// TIA Portal V20 export
FUNCTION_BLOCK "Simulation"   // FB25, LAD
// stored: MemoryReserve 100, Namespace Unit1.Em5, SetENOAutomatically false
   VAR_INPUT
      simulation { ExternalAccessible := 'False'; ExternalVisible := 'False'; ExternalWritable := 'False'} : Bool;
   END_VAR
   VAR
      instMainPnPActuator { ExternalAccessible := 'False'; ExternalVisible := 'False'; ExternalWritable := 'False'} : Array[0..9] of "LER_SimActuator";
      instAlignTableActuator { ExternalAccessible := 'False'; ExternalVisible := 'False'; ExternalWritable := 'False'} : Array[0..9] of "LER_SimActuator";
      instNgPnPActuator { ExternalAccessible := 'False'; ExternalVisible := 'False'; ExternalWritable := 'False'} : Array[0..9] of "LER_SimActuator";
   END_VAR
   VAR_TEMP   // added for the SCL form of the ladder/FBD networks
      _w1 : Bool;
   END_VAR
BEGIN

REGION Network 1: Main P&P Two Way Actuator
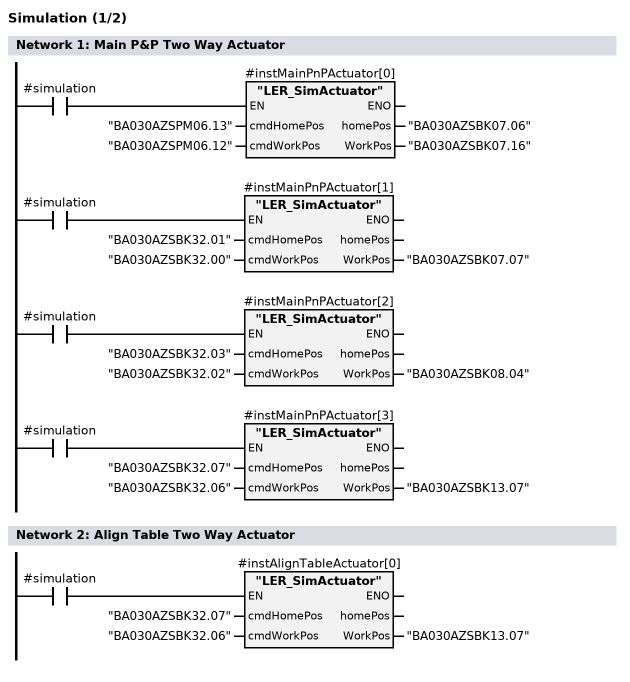
   RUNG wire#powerrail
      Contact( #simulation )
      #instMainPnPActuator[0](cmdHomePos := "BA030AZSPM06.13", cmdWorkPos := "BA030AZSPM06.12", homePos => "BA030AZSBK07.06", WorkPos => "BA030AZSBK07.16")
   END_RUNG
   RUNG wire#powerrail
      Contact( #simulation )
      #instMainPnPActuator[1](cmdHomePos := "BA030AZSBK32.01", cmdWorkPos := "BA030AZSBK32.00", homePos =>, WorkPos => "BA030AZSBK07.07")
   END_RUNG
   RUNG wire#powerrail
      Contact( #simulation )
      #instMainPnPActuator[2](cmdHomePos := "BA030AZSBK32.03", cmdWorkPos := "BA030AZSBK32.02", homePos =>, WorkPos => "BA030AZSBK08.04")
   END_RUNG
   RUNG wire#powerrail
      Contact( #simulation )
      #instMainPnPActuator[3](cmdHomePos := "BA030AZSBK32.07", cmdWorkPos := "BA030AZSBK32.06", homePos =>, WorkPos => "BA030AZSBK13.07")
   END_RUNG
   // the same network as SCL:
   IF #simulation THEN
       #instMainPnPActuator[0](cmdHomePos := "BA030AZSPM06.13",   // "LER_SimActuator"
                               cmdWorkPos := "BA030AZSPM06.12",
                               homePos => "BA030AZSBK07.06",
                               WorkPos => "BA030AZSBK07.16");
       #instMainPnPActuator[1](cmdHomePos := "BA030AZSBK32.01",   // "LER_SimActuator"
                               cmdWorkPos := "BA030AZSBK32.00",
                               WorkPos => "BA030AZSBK07.07");
       #instMainPnPActuator[2](cmdHomePos := "BA030AZSBK32.03",   // "LER_SimActuator"
                               cmdWorkPos := "BA030AZSBK32.02",
                               WorkPos => "BA030AZSBK08.04");
       #instMainPnPActuator[3](cmdHomePos := "BA030AZSBK32.07",   // "LER_SimActuator"
                               cmdWorkPos := "BA030AZSBK32.06",
                               WorkPos => "BA030AZSBK13.07");
   END_IF;
END_REGION

REGION Network 2: Align Table Two Way Actuator
   RUNG wire#powerrail
      Contact( #simulation )
      #instAlignTableActuator[0](cmdHomePos := "BA030AZSBK32.07", cmdWorkPos := "BA030AZSBK32.06", homePos =>, WorkPos => "BA030AZSBK13.07")
   END_RUNG
   // the same network as SCL:
   IF #simulation THEN
       #instAlignTableActuator[0](cmdHomePos := "BA030AZSBK32.07",   // "LER_SimActuator"
                               cmdWorkPos := "BA030AZSBK32.06",
                               WorkPos => "BA030AZSBK13.07");
   END_IF;
END_REGION

REGION Network 3: NG P&P Two Way Actuator
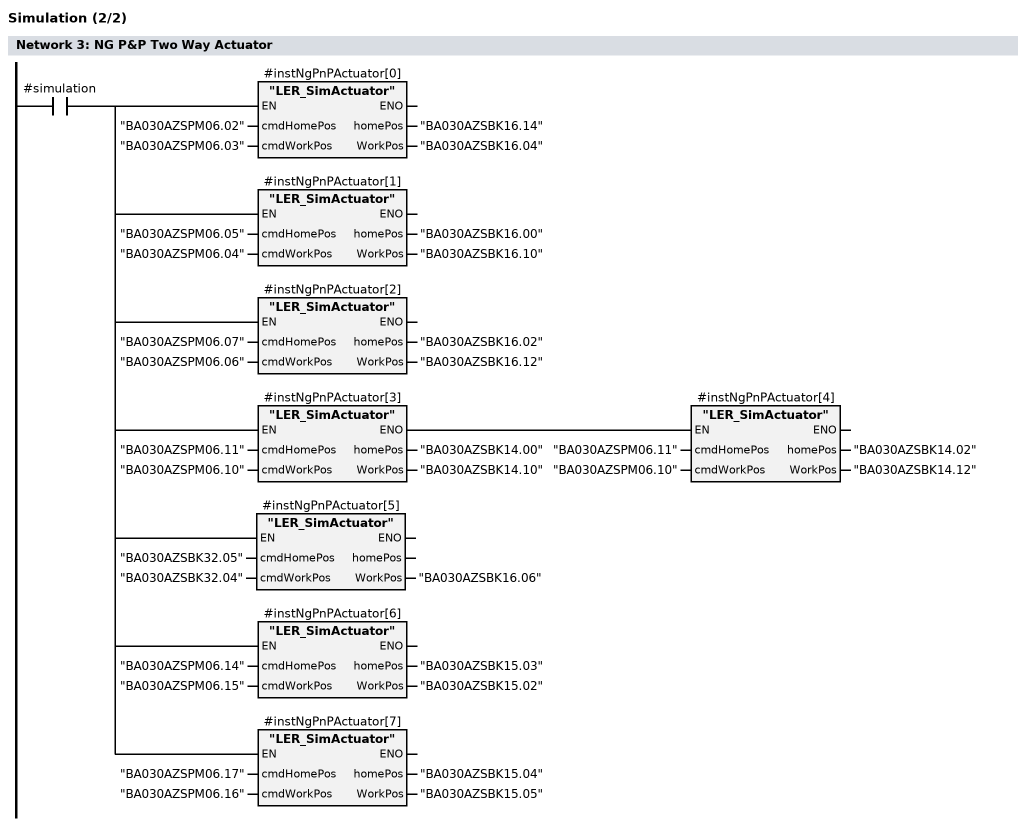
   RUNG wire#powerrail
      Contact( #simulation )
      wire#w1
      #instNgPnPActuator[0](cmdHomePos := "BA030AZSPM06.02", cmdWorkPos := "BA030AZSPM06.03", homePos => "BA030AZSBK16.14", WorkPos => "BA030AZSBK16.04")
   END_RUNG
   RUNG wire#w1
      #instNgPnPActuator[1](cmdHomePos := "BA030AZSPM06.05", cmdWorkPos := "BA030AZSPM06.04", homePos => "BA030AZSBK16.00", WorkPos => "BA030AZSBK16.10")
   END_RUNG
   RUNG wire#w1
      #instNgPnPActuator[2](cmdHomePos := "BA030AZSPM06.07", cmdWorkPos := "BA030AZSPM06.06", homePos => "BA030AZSBK16.02", WorkPos => "BA030AZSBK16.12")
   END_RUNG
   RUNG wire#w1
      #instNgPnPActuator[3](cmdHomePos := "BA030AZSPM06.11", cmdWorkPos := "BA030AZSPM06.10", homePos => "BA030AZSBK14.00", WorkPos => "BA030AZSBK14.10")
      #instNgPnPActuator[4](cmdHomePos := "BA030AZSPM06.11", cmdWorkPos := "BA030AZSPM06.10", homePos => "BA030AZSBK14.02", WorkPos => "BA030AZSBK14.12")
   END_RUNG
   RUNG wire#w1
      #instNgPnPActuator[5](cmdHomePos := "BA030AZSBK32.05", cmdWorkPos := "BA030AZSBK32.04", homePos =>, WorkPos => "BA030AZSBK16.06")
   END_RUNG
   RUNG wire#w1
      #instNgPnPActuator[6](cmdHomePos := "BA030AZSPM06.14", cmdWorkPos := "BA030AZSPM06.15", homePos => "BA030AZSBK15.03", WorkPos => "BA030AZSBK15.02")
   END_RUNG
   RUNG wire#w1
      #instNgPnPActuator[7](cmdHomePos := "BA030AZSPM06.17", cmdWorkPos := "BA030AZSPM06.16", homePos => "BA030AZSBK15.04", WorkPos => "BA030AZSBK15.05")
   END_RUNG
   // the same network as SCL:
   IF #simulation THEN
       #instNgPnPActuator[0](cmdHomePos := "BA030AZSPM06.02",   // "LER_SimActuator"
                             cmdWorkPos := "BA030AZSPM06.03",
                             homePos => "BA030AZSBK16.14",
                             WorkPos => "BA030AZSBK16.04");
       #instNgPnPActuator[1](cmdHomePos := "BA030AZSPM06.05",   // "LER_SimActuator"
                             cmdWorkPos := "BA030AZSPM06.04",
                             homePos => "BA030AZSBK16.00",
                             WorkPos => "BA030AZSBK16.10");
       #instNgPnPActuator[2](cmdHomePos := "BA030AZSPM06.07",   // "LER_SimActuator"
                             cmdWorkPos := "BA030AZSPM06.06",
                             homePos => "BA030AZSBK16.02",
                             WorkPos => "BA030AZSBK16.12");
   END_IF;
   #instNgPnPActuator[3](EN := #simulation,   // "LER_SimActuator"
                         cmdHomePos := "BA030AZSPM06.11",
                         cmdWorkPos := "BA030AZSPM06.10",
                         homePos => "BA030AZSBK14.00",
                         WorkPos => "BA030AZSBK14.10",
                         ENO => #_w1);
   IF #_w1 THEN
       #instNgPnPActuator[4](cmdHomePos := "BA030AZSPM06.11",   // "LER_SimActuator"
                             cmdWorkPos := "BA030AZSPM06.10",
                             homePos => "BA030AZSBK14.02",
                             WorkPos => "BA030AZSBK14.12");
   END_IF;
   IF #simulation THEN
       #instNgPnPActuator[5](cmdHomePos := "BA030AZSBK32.05",   // "LER_SimActuator"
                             cmdWorkPos := "BA030AZSBK32.04",
                             WorkPos => "BA030AZSBK16.06");
       #instNgPnPActuator[6](cmdHomePos := "BA030AZSPM06.14",   // "LER_SimActuator"
                             cmdWorkPos := "BA030AZSPM06.15",
                             homePos => "BA030AZSBK15.03",
                             WorkPos => "BA030AZSBK15.02");
       #instNgPnPActuator[7](cmdHomePos := "BA030AZSPM06.17",   // "LER_SimActuator"
                             cmdWorkPos := "BA030AZSPM06.16",
                             homePos => "BA030AZSBK15.04",
                             WorkPos => "BA030AZSBK15.05");
   END_IF;
END_REGION
END_FUNCTION_BLOCK
